// TIA Portal V16 export
// export: Created 2021-03-05T14:22:12.2245166Z, ExportSetting WithDefaults, DisplayName Totally Integrated Automation Portal, DisplayVersion V16, DisplayName TIA Portal Version Control Interface, DisplayVersion V16, DisplayName TIA Portal Openness, DisplayVersion V16, DisplayName SINAMICS Startdrive Advanced, DisplayVersion V16, DisplayName SINAMICS Startdrive G130, G150, S120, S150, SINAMICS MV, S210, DisplayVersion V16, DisplayName SINAMICS Startdrive G110M, G120, G120C, G120D, G120P, DisplayVersion V16, DisplayName STEP 7 Professional, DisplayVersion V16, DisplayName STEP 7 Safety, DisplayVersion V16, DisplayName WinCC Professional, DisplayVersion V16
FUNCTION_BLOCK "fbRackFertigation"   // FB1, LAD
{ S7_Optimized_Access := 'TRUE' }
VERSION : 0.1
// stored: AutoNumber true, IsIECCheckEnabled false, IsRetainMemResEnabled false, MemoryReserve 100, SetENOAutomatically false, UDAEnableTagReadback false
   VAR_INPUT
      arrAI : Array[1.."NUM_AI_RACK"] of Int;
      AI AT arrAI : Array[1.."NUM_AI_RACK"] of Int;
   END_VAR
   VAR_OUTPUT
      arrDQ : Array[1.."NUM_DQ_RACK"] of Bool;
      DQ AT arrDQ : "udtRackDQ";
   END_VAR
   VAR RETAIN
      Controls : Struct
         Flood_Duration : LInt := 5;   // Minutes - not currently used, but here for when rack-level confgurations are desired over shelf-level
         Flood_Interval : Int := 120;   // Minutes - see above
         Num_Shelves : Int := 6;
         ROCommand : Bool;
         DischargeCommand : Bool;
         RunMode : Int;   // 0: off, 2: auto(flood/soak/drain) 3: discharge
         ReservoirLowLimit : Real := 25.0;   // Liters
         ReservoirUpperLimit : Real := 60.0;   // Liters
      END_STRUCT;
      Status : Struct
         Active_Shelf : Int := -1;
         Last_Flood { S7_SetPoint := 'True'} : Date_And_Time := DT#2015-01-01-00:00:00;   // not currently used, but here for when rack-level confgurations are desired over shelf-level
      END_STRUCT;
      AI_Reservoir_Level { S7_SetPoint := 'True'} : "udtAnalogInput";
   END_VAR
   VAR
      DQ_RO_Solenoid : "udtDigitalOutput";
      DQ_Discharge_Solenoid : "udtDigitalOutput";
      ShelvesFertigation : Array[1.."NUM_SHELVES_PER_RACK"] of "fbShelfFertigation";
   END_VAR
   VAR_TEMP
      i : Int;
      current_date_time : Date_And_Time;
      retval : Int;
      td_diff : Time;
      minutes_diff : LInt;
      current_date : LDT;
      current_time : LTime_Of_Day;
      shelf_last_date : LDT;
      day_diff : LTime;
      shelf_last_time : LTime_Of_Day;
      flood_time : Time;
      active_shelves : Int;
      j : Int;
   END_VAR
   VAR CONSTANT
      drain_time : Time := T#300S;
   END_VAR
   // // AI_Reservoir_Level.rActual : Liters
BEGIN

REGION Network 1 (SCL): map AI
   #AI_Reservoir_Level.rRawValue := #arrAI[1];
   #AI_Reservoir_Level.rActual := "fcAnalogInput"(iInRawValue := #AI_Reservoir_Level.rRawValue,
                                                  rLowCalibration := #AI_Reservoir_Level.rLowCalibration,
                                                  rHighCalibration := #AI_Reservoir_Level.rHighCalibration);
END_REGION

REGION Network 2 (SCL)

   REGION 0: OFF 
       // deactivate all shelves
       IF #Controls.RunMode = 0 THEN
           FOR #i := 1 TO #Controls.Num_Shelves DO
               #ShelvesFertigation[#i].Status.Active := False;
               #Status.Active_Shelf := -1;
           END_FOR;

           #Controls.ROCommand := False;
           #Controls.DischargeCommand := False;
       END_IF;

   END_REGION



   REGION 2: AUTO

       IF #Controls.RunMode = 2 THEN

           IF #AI_Reservoir_Level.rActual < #Controls.ReservoirUpperLimit AND #Status.Active_Shelf = -1 THEN
               // do not fill reservoir while flood-soak-drain sequence in progress
               #Controls.ROCommand := True;
           ELSE
               #Controls.ROCommand := False;
           END_IF;

           #Controls.DischargeCommand := False;

           IF NOT #Controls.ROCommand THEN
               // do not execute shelf flood-soak-drain logic while filling reservoir

               FOR #i := 1 TO #Controls.Num_Shelves DO
                   // get current date and time
                   #retval := RD_LOC_T(#current_date_time);
                   #current_date := DT_TO_LDT(#current_date_time);
                   #current_time := DT_TO_LTOD(#current_date_time);

                   // get last time rack flood loop ran 
                   #shelf_last_date := DT_TO_LDT(#ShelvesFertigation[#i].Controls.Last_Flood);
                   #shelf_last_time := DT_TO_LTOD(#ShelvesFertigation[#i].Controls.Last_Flood);

                   // calculate difference in seconds
                   #day_diff := T_DIFF(IN1 := #current_date, IN2 := #shelf_last_date);
                   #minutes_diff := LTIME_TO_LINT(#day_diff);
                   #minutes_diff := (#minutes_diff / 1000000) / 60000;

                   IF #minutes_diff > #Controls.Flood_Interval
                   THEN
                       IF #Status.Active_Shelf = -1 AND #ShelvesFertigation[#i].Status.Active THEN
                           #Status.Active_Shelf := #i;
                       END_IF;
                   END_IF;

                   IF #ShelvesFertigation[#i].Status.Finished AND #i = #Status.Active_Shelf THEN
                       #ShelvesFertigation[#i].Status.Finished := 0;
                       #Status.Active_Shelf := -1; // next shelf's turn...
                   END_IF;

               END_FOR;
           END_IF;
       END_IF;


   END_REGION


   REGION 3: Discharge
       // dump reservoir contents to drain, then switch off

       IF #Controls.RunMode = 3 THEN

           #Controls.ROCommand := False;

           IF #AI_Reservoir_Level.rActual > #Controls.ReservoirLowLimit THEN
               #Controls.DischargeCommand := TRUE;
           ELSE
               #Controls.DischargeCommand := FALSE;
               #Controls.RunMode := 0; //off
               FOR #i := 1 TO #Controls.Num_Shelves DO
                   #ShelvesFertigation[#i].Status.Active := False;
                   #Status.Active_Shelf := -1;
               END_FOR;
           END_IF;
       END_IF;


   END_REGION
END_REGION

REGION Network 3 (SCL): Execute shelf fertigation logic
   FOR #i := 1 TO #Controls.Num_Shelves DO
       #ShelvesFertigation[#i](activeShelf := #Status.Active_Shelf,
                               shelfNumber := #i,
                               arrDQ => #ShelvesFertigation[#i].arrDQ,
                               ReservoirLevel := #AI_Reservoir_Level.rActual,
                               RunMode := #Controls.RunMode
       );
   END_FOR;
END_REGION

REGION Network 4 (SCL)
   #DQ.Q_RO_BV := "fcDigitalOutput"(bInAutoVal := #Controls.ROCommand, InOutUdt := #DQ_RO_Solenoid);
   #DQ.Q_Discharge_BV := "fcDigitalOutput"(bInAutoVal := #Controls.DischargeCommand, InOutUdt := #DQ_Discharge_Solenoid);
END_REGION
END_FUNCTION_BLOCK
